FUNCTION_BLOCK fb_base
VAR_INPUT
END_VAR
VAR_OUTPUT
END_VAR
VAR
END_VAR

END_FUNCTION_BLOCK

(* stored: Version 1.1.0.1, ProductVersion 3.1.4024.12
   POU fb_base: Id {13f26e08-97c7-4564-bd47-e569329f30de}, SpecialFunc None *)
